FUNCTION_BLOCK FB_MotionDriveStateMachine_TestDouble IMPLEMENTS I_MotionDriveStateMachine
VAR
END_VAR

{warning 'Add property implementation'}
PROPERTY Idling : BOOL
GET
END_GET
END_PROPERTY

PROPERTY MoveState : E_MOVESTATE
GET
END_GET
END_PROPERTY

METHOD StateMachine
VAR_INPUT
    Error	: BOOL;
END_VAR
END_METHOD

PROPERTY WatchDogStatus : BOOL
GET
END_GET
END_PROPERTY

PROPERTY WatchDogTimeOut : BOOL
GET
END_GET
END_PROPERTY

END_FUNCTION_BLOCK

(* stored: Version 1.1.0.1
   POU FB_MotionDriveStateMachine_TestDouble: Id {bd4c0fda-2c0f-4d99-bff0-ed190100a01c}, SpecialFunc None
   Property Idling: Id {4d1775a0-7b36-4458-b6bc-000998f7c70b}
   Get Get: Id {0ae0842e-3354-4ebf-a230-b2374daccdd0}
   Property MoveState: Id {5b8ab468-efd2-474c-930c-53db7f21c503}
   Get Get: Id {d8032f69-63db-4d74-bbc2-c680fd7b80fa}
   Method StateMachine: Id {53a2f700-2d7e-4499-830f-475a67ac2b82}
   Property WatchDogStatus: Id {e6fb2611-cf62-410c-b73d-4c60b0873c32}
   Get Get: Id {6302b0ad-2cc0-4385-83f3-ee776beb4493}
   Property WatchDogTimeOut: Id {18a85cf8-05cc-4f4c-b8a1-59a6774c4d9d}
   Get Get: Id {0ada9824-d6e4-439b-a047-2c42f8f82b99} *)
